// TIA Portal project "test" (V20)

(* hardware
DEVICE "S7-1200 station_1"  S7-1200 Station
   slot 0: "Rack_0"  S7-1200 Rack  Rack  V1.0
   slot 1: "PLC_1"  CPU 1211C DC/DC/DC  6ES7 211-1AE40-0XB0  V4.7
*)

// ===== PLC "PLC_1"  CPU 1211C DC/DC/DC =====

VAR_GLOBAL   // PLC tag table "Default tag table"
   "In_1" AT %I0.0 : Bool;
   "Out1" AT %Q0.0 : Bool;
   "NC_1" AT %I0.1 : Bool;
   "NC_out" AT %Q0.1 : Bool;
   "P1" AT %I0.2 : Bool;
   "P2" AT %I0.3 : Bool;
   "P_out" AT %Q0.2 : Bool;
   "S1" AT %I0.4 : Bool;
   "S2" AT %I0.5 : Bool;
   "S_out" AT %Q0.3 : Bool;
END_VAR

ORGANIZATION_BLOCK "Main"   // OB1, LAD, ProgramCycle
TITLE = "Main Program Sweep (Cycle)"
{ S7_Optimized_Access := 'TRUE' }
VERSION : 0.1
   VAR_INPUT
      Initial_Call : Bool;   // Initial call of this OB
      Remanence : Bool;   // =True, if remanent data are available
   END_VAR
BEGIN

REGION Network 1
   // Normalmente Abierto
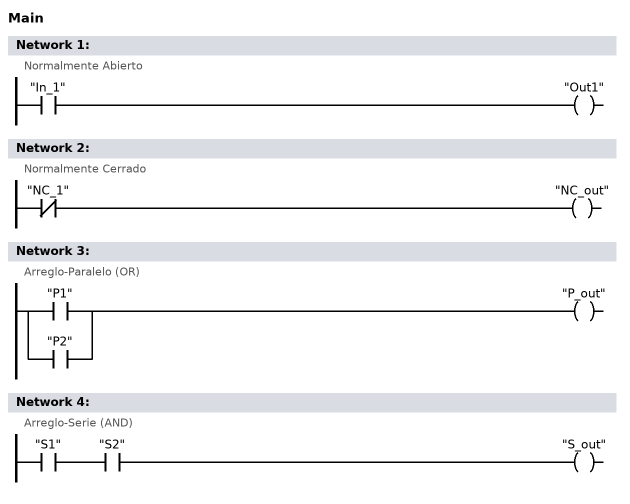
   RUNG wire#powerrail
      Contact( "In_1" )
      Coil( "Out1" )
   END_RUNG
   // the same network as SCL:
   "Out1" := "In_1";
END_REGION

REGION Network 2
   // Normalmente Cerrado
   RUNG wire#powerrail
      I_Contact( "NC_1" )
      Coil( "NC_out" )
   END_RUNG
   // the same network as SCL:
   "NC_out" := NOT "NC_1";
END_REGION

REGION Network 3
   // Arreglo-Paralelo (OR)
   RUNG wire#powerrail
      Contact( "P1" )
      wire#w1
      Coil( "P_out" )
   END_RUNG
   RUNG wire#powerrail
      Contact( "P2" )
   END_RUNG wire#w1
   // the same network as SCL:
   "P_out" := "P1" OR "P2";
END_REGION

REGION Network 4
   // Arreglo-Serie (AND)
   RUNG wire#powerrail
      Contact( "S1" )
      Contact( "S2" )
      Coil( "S_out" )
   END_RUNG
   // the same network as SCL:
   "S_out" := "S1" AND "S2";
END_REGION
END_ORGANIZATION_BLOCK